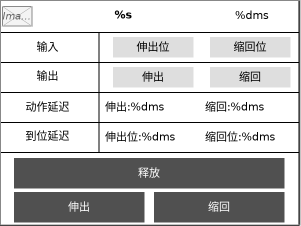
VISUALIZATION Cyliner1  // 301x226
VAR_INPUT
	System:							REFERENCE TO ST_System;
	Cylinder:						REFERENCE TO ST_Cylinder;
	CylinderData:					REFERENCE TO ST_CylinderData;
END_VAR
    RoundedRectangle (-1,111 300x115)
    RoundedRectangle (-1,0 300x115)
    Rectangle (-1,34 300x115)
    Line (-1,32) (299,32)
    Rectangle (34,3 179x24), "%s", text variable: Cylinder.arrInfo[System.stMode.eLanguage].sName, input disabled if: Cylinder.stLock.bShield
    Rectangle (217,3 70x25), "%dms", text variable: CylinderData.iAlarmTime, input disabled if: Cylinder.stLock.bShield
        OnMouseClick: write the text variable via VisuDialogs.Numpad
    Line (-1,62) (299,62)
    Line (-1,92) (299,92)
    Label (0,32 95x30), "输入"
    Label (0,61 95x30), "输出"
    Line (99,152) (99,32)
    RoundedRectangle (113,37 80x20), "伸出位", colour toggle: Cylinder.stInput.bWork, input disabled if: Cylinder.stLock.bShield
    RoundedRectangle (210,37 80x20), "缩回位", colour toggle: Cylinder.stInput.bHome, input disabled if: Cylinder.stLock.bShield
    RoundedRectangle (113,67 80x20), "伸出", colour toggle: Cylinder.stOutput.bWork, input disabled if: Cylinder.stLock.bShield
    RoundedRectangle (210,67 80x20), "缩回", colour toggle: Cylinder.stOutput.bHome, input disabled if: Cylinder.stLock.bShield
    RoundedRectangle (14,158 270x30), "释放", colour toggle: Cylinder.stLock.bOff OR Cylinder.stLock.bAll, input disabled if: Cylinder.stLock.bShield
        tap Cylinder.stControl.stOffRequest.bManual
    RoundedRectangle (14,192 130x30), "伸出", colour toggle: Cylinder.stLock.bWork OR Cylinder.stLock.bAll, input disabled if: Cylinder.stLock.bShield
        tap Cylinder.stControl.stWorkRequest.bManual
    RoundedRectangle (154,192 130x30), "缩回", colour toggle: Cylinder.stLock.bHome OR Cylinder.stLock.bAll, input disabled if: Cylinder.stLock.bShield
        tap Cylinder.stControl.stHomeRequest.bManual
    Line (299,154) (299,23)
    Line (-1,152) (-1,19)
    Image (2,6 30x20), image: ImagePool.Cylinder1
    Line (-1,122) (299,122)
    Line (-1,152) (299,152)
    Label (0,92 95x30), "动作延迟"
    Label (0,121 95x30), "到位延迟"
    RoundedRectangle (102,94 95x26), "伸出:%dms", text variable: CylinderData.iWorkRequestTime, input disabled if: Cylinder.stLock.bShield
        OnMouseClick: write the text variable via Default
    RoundedRectangle (202,94 95x26), "缩回:%dms", text variable: CylinderData.iHomeRequestTime, input disabled if: Cylinder.stLock.bShield
        OnMouseClick: write the text variable via Default
    RoundedRectangle (102,124 95x26), "伸出位:%dms", text variable: CylinderData.iWorkDone, input disabled if: Cylinder.stLock.bShield
        OnMouseClick: write the text variable via Default
    RoundedRectangle (202,124 95x26), "缩回位:%dms", text variable: CylinderData.iHomeDone, input disabled if: Cylinder.stLock.bShield
        OnMouseClick: write the text variable via Default
END_VISUALIZATION

(* stored: Version 1.1.0.1, ProductVersion 3.1.4024.4
   Visu Cyliner1: Id {c0efdf03-6af8-4d7f-90e7-cbf1734bcc96} *)
